PROGRAM MAIN
VAR
	nServoSpeed : DINT;
	
	AxisB : AXIS_REF;
	bSafetyCondition: BOOL;
	McPower : MC_Power;
	McReset : MC_Reset;
	McJogging : MC_Jog;
	McVelo : MC_MoveVelocity;
	McStop : MC_Stop;
	bVirtualMoveVelo : BOOL;
	bVirtualStop : BOOL;
	
	
	iState : INT; // my state
	nLastThrottle : INT;
END_VAR

bSafetyCondition:= PRG_Safety.fbTsConnection_EL2904.stTsSlaveInfo.bChannel1;

IF (IO.bButton1 OR bVirtualMoveVelo) AND bSafetyCondition THEN
	IO.bLed1:= TRUE;
END_IF

IF (IO.bButton2 OR bVirtualStop) OR NOT bSafetyCondition THEN
	IO.bLed1:=FALSE;
END_IF

IO.nPotentiometer := IO.nSpeedCmd;
nServoSpeed := F_Scale(nAIn:= IO.nSpeedCmd, 100.0, 2800.0, 0, 32767);

// Drive Control
AxisB.ReadStatus();
McPower(Axis:=AxisB,Enable:= TRUE, Enable_Positive:= TRUE, Enable_Negative:=TRUE);
McReset(Axis:=AxisB);
McJogging(Axis:=AxisB);

CASE iState OF
	0:
		iState:= 10; //initial
	10: // Start drive reset
		IF McPower.Status THEN
			McReset(Axis:= AxisB, Execute:=TRUE);
			IF McReset.Done THEN
				iState:=20;
			ELSIF McReset.Error THEN
				iState:=-999;		
			END_IF
		END_IF
			
	20: // Wait for drive to reset
		IF McPower.Status THEN
			iState:=30;
		END_IF
	30: // Wait for drive command
		//McJogging(Axis:=AxisB, JogForward := IO.bLed1);
		McVelo(
			Axis:= AxisB,
			Execute:= IO.bLed1 AND IO.nSpeedCmd <> nLastThrottle,
			Velocity:= nServoSpeed,
			Acceleration := 10000,
			Deceleration := 10000,
			Jerk := 10000000,
			Direction:= MC_DIRECTION.MC_Positive_Direction
		);
		IF NOT IO.bLed1 OR NOT bSafetyCondition THEN
			McVelo(Axis:=AxisB, Execute:= FALSE);
			iState:=900;
		END_IF
		nLastThrottle := IO.nSpeedCmd;
	900: // Stop Servo
		McStop(Axis:= AxisB, Execute:= TRUE);
		IF IO.bLed1 AND bSafetyCondition THEN
			McStop(Axis:= AxisB, Execute:= FALSE);
			iState:=30;
		END_IF
	-999: // Handle error
END_CASE


PRG_Safety();

END_PROGRAM

(* stored: Version 1.1.0.1, ProductVersion 3.1.4024.12
   POU MAIN: Id {c68557e9-d255-42aa-8e04-c3eae67d9a27}, SpecialFunc None *)
